// TIA Portal V17 export
// export: Created 2024-08-26T21:07:22.2983378Z, ExportSetting WithDefaults, DisplayName Totally Integrated Automation Portal, DisplayVersion V17 Update 7, DisplayName TIA Portal Openness, DisplayVersion V17 Update 7, DisplayName TIA Portal Version Control Interface, DisplayVersion V17, DisplayName SINAMICS Startdrive Advanced, DisplayVersion V17 SP2, DisplayName SINAMICS Startdrive G110M, G120, G120C, G120D, G120P, G115D, DisplayVersion V17 SP2, DisplayName SINAMICS Startdrive G130, G150, S120, S150, SINAMICS MV, S210, DisplayVersion V17 SP2, DisplayName STEP 7 Professional, DisplayVersion V17 Update 7, DisplayName STEP 7 Safety, DisplayVersion V17 Update 6, DisplayName WinCC Advanced / Unified PC, DisplayVersion V17 Update 7
VAR_GLOBAL   // PLC tag table "permissionMemory"
   MaintenacePermission AT %M4.4 : Bool;
   adminPermission AT %M4.0 : Bool;
   lgPermission AT %M4.5 : Bool;
   gapLeaderUser AT %M4.3 : Bool;
   editingPermission AT %M4.1 : Bool;
   confirmStandby AT %M5.7 : Bool;
   cancelMovement AT %M8.0 : Bool;
END_VAR
